// TIA Portal V20 export
TYPE "typeEm1Commands"
// stored: Access Published, Namespace Unit1
   STRUCT
      jobinterface { ExternalWritable := 'False'} : "Unit1.typeEm1CommandsJobInterface";
   END_STRUCT;
END_TYPE
